// TIA Portal V17 export
// export: Created 2024-01-30T08:49:16.7759616Z, ExportSetting WithDefaults, DisplayName Totally Integrated Automation Portal, DisplayVersion V17 Update 6, DisplayName TIA Portal Openness, DisplayVersion V17 Update 6, DisplayName TIA Portal Version Control Interface, DisplayVersion V17, DisplayName STEP 7 Professional, DisplayVersion V17 Update 6, DisplayName STEP 7 Safety, DisplayVersion V17 Update 6, DisplayName WinCC Advanced, DisplayVersion V17 Update 6
VAR_GLOBAL   // PLC tag table "Standard-Variablentabelle"
   "LK-H057_01" AT %IW322 : Word;
   "LK-H057_02" AT %IW324 : Word;
   Tag_1 AT %ID70 : Real;
   Tag_2 AT %ID74 : DWord;
   Clock_Byte AT %MB0 : Byte;
   Clock_10Hz AT %M0.0 : Bool;
   Clock_5Hz AT %M0.1 : Bool;
   "Clock_2.5Hz" AT %M0.2 : Bool;
   Clock_2Hz AT %M0.3 : Bool;
   "Clock_1.25Hz" AT %M0.4 : Bool;
   Clock_1Hz AT %M0.5 : Bool;
   "Clock_0.625Hz" AT %M0.6 : Bool;
   "Clock_0.5Hz" AT %M0.7 : Bool;
   RS232_SEND_Req AT %M100.0 : Bool;
   Tag_3 AT %M100.1 : Bool;
   Tag_4 AT %M100.2 : Bool;
   RS232_Send AT %M100.3 : Bool;
   Data_log_StartStop AT %M100.4 : Bool;
   Tag_5 AT %M100.5 : Bool;
   Tag_6 AT %M100.6 : Bool;
   Tag_7 AT %M100.7 : Bool;
   Tag_8 AT %M101.0 : Bool;
   Tag_9 AT %M101.1 : Bool;
   FALSE AT %M101.2 : Bool;
   Tag_10 AT %M200.0 : Bool;
   Tag_11 AT %M200.1 : Bool;
   Tag_12 AT %M200.2 : Bool;
END_VAR
